PROGRAM MAIN
VAR
END_VAR

Motion();

END_PROGRAM

(* stored: Version 1.1.0.1, ProductVersion 3.1.4024.12
   POU MAIN: Id {a598916d-876e-499b-ab6a-e0adb19e3e4a}, SpecialFunc None *)
